// TIA Portal V18 export
VAR_GLOBAL   // PLC tag table "Default tag table"
   CS_Drive_PL_Actor_Interface_AddressIn AT %I50.0 : "PD_TEL105_IN";
   CS_Drive_PL_Actor_Interface_AddressOut AT %Q50.0 : "PD_TEL105_OUT";
   CS_Drive_PP_Actor_Interface_AddressIn AT %I18.0 : "PD_TEL105_IN";
   CS_Drive_PP_Actor_Interface_AddressOut AT %Q18.0 : "PD_TEL105_OUT";
   CS_Drive_TL_Actor_Interface_AddressIn AT %I102.0 : "PD_TEL105_IN";
   CS_Drive_TL_Actor_Interface_AddressOut AT %Q102.0 : "PD_TEL105_OUT";
   CS_Drive_TP_Actor_Interface_AddressIn AT %I76.0 : "PD_TEL105_IN";
   CS_Drive_TP_Actor_Interface_AddressOut AT %Q76.0 : "PD_TEL105_OUT";
   ST23_PAL_Down AT %Q900.0 : Bool;
   ST23_PAL_Up AT %Q900.1 : Bool;
   ST23_MOD1_Up AT %Q900.2 : Bool;
   ST23_MOD2_Up AT %Q900.3 : Bool;
   ST23_MOD3_Up AT %Q900.4 : Bool;
   ST24_PAL_Down AT %Q900.5 : Bool;
   ST24_PAL_Up AT %Q900.6 : Bool;
   ST24_MOD1_Up AT %Q900.7 : Bool;
   ST24_MOD2_Up AT %Q901.0 : Bool;
   ST24_MOD3_Up AT %Q901.1 : Bool;
   ST25_PAL_Down AT %Q901.2 : Bool;
   ST25_PAL_Up AT %Q901.3 : Bool;
   ST25_MOD1_Up AT %Q901.4 : Bool;
   ST25_MOD2_Up AT %Q901.5 : Bool;
   ST25_MOD3_Up AT %Q901.6 : Bool;
   Reserve AT %Q901.7 : Bool;
   ST23_MOD1_Sen11 AT %I900.0 : Bool;
   ST23_MOD1_Sen12 AT %I900.1 : Bool;
   ST23_MOD1_Sen21 AT %I900.2 : Bool;
   ST23_MOD1_Sen22 AT %I900.3 : Bool;
   ST23_MOD2_Sen11 AT %I900.4 : Bool;
   ST23_MOD2_Sen12 AT %I900.5 : Bool;
   ST23_MOD2_Sen21 AT %I900.6 : Bool;
   ST23_MOD2_Sen22 AT %I900.7 : Bool;
   ST23_MOD3_Sen11 AT %I901.0 : Bool;
   ST23_MOD3_Sen12 AT %I901.1 : Bool;
   ST23_MOD3_Sen21 AT %I901.2 : Bool;
   ST23_MOD3_Sen22 AT %I901.3 : Bool;
   ST23_PAL_Sen11 AT %I901.4 : Bool;
   ST23_PAL_Sen12 AT %I901.5 : Bool;
   ST23_PAL_Sen21 AT %I901.6 : Bool;
   ST23_PAL_Sen22 AT %I901.7 : Bool;
   ST24_MOD1_Sen11 AT %I902.0 : Bool;
   ST24_MOD1_Sen12 AT %I902.1 : Bool;
   ST24_MOD1_Sen21 AT %I902.2 : Bool;
   ST24_MOD1_Sen22 AT %I902.3 : Bool;
   ST24_MOD2_Sen11 AT %I902.4 : Bool;
   ST24_MOD2_Sen12 AT %I902.5 : Bool;
   ST24_MOD2_Sen21 AT %I902.6 : Bool;
   ST24_MOD2_Sen22 AT %I902.7 : Bool;
   ST24_MOD3_Sen11 AT %I903.0 : Bool;
   ST24_MOD3_Sen12 AT %I903.1 : Bool;
   ST24_MOD3_Sen21 AT %I903.2 : Bool;
   ST24_MOD3_Sen22 AT %I903.3 : Bool;
   ST24_PAL_Sen11 AT %I903.4 : Bool;
   ST24_PAL_Sen12 AT %I903.5 : Bool;
   ST24_PAL_Sen21 AT %I903.6 : Bool;
   ST24_PAL_Sen22 AT %I903.7 : Bool;
   ST23_Rol_Up AT %Q902.0 : Bool;
   ST24_Rol_Up AT %Q902.1 : Bool;
   ST25_Rol_Up AT %Q902.2 : Bool;
   ST25_MOD1_Sen11 AT %I904.0 : Bool;
   ST25_MOD1_Sen12 AT %I904.1 : Bool;
   ST25_MOD1_Sen21 AT %I904.2 : Bool;
   ST25_MOD1_Sen22 AT %I904.3 : Bool;
   ST25_MOD2_Sen11 AT %I904.4 : Bool;
   ST25_MOD2_Sen12 AT %I904.5 : Bool;
   ST25_MOD2_Sen21 AT %I904.6 : Bool;
   ST25_MOD2_Sen22 AT %I904.7 : Bool;
   ST25_MOD3_Sen11 AT %I905.0 : Bool;
   ST25_MOD3_Sen12 AT %I905.1 : Bool;
   ST25_MOD3_Sen21 AT %I905.2 : Bool;
   ST25_MOD3_Sen22 AT %I905.3 : Bool;
   ST25_PAL_Sen11 AT %I905.4 : Bool;
   ST25_PAL_Sen12 AT %I905.5 : Bool;
   ST25_PAL_Sen21 AT %I905.6 : Bool;
   ST25_PAL_Sen22 AT %I905.7 : Bool;
   "90" AT %Q0.0 : Bool;
   Estop_SS2_ChA AT %I915.0 : Bool;
   Estop_SS2_ChB AT %I915.4 : Bool;
   ST23_25_Y0 AT %Q910.0 : Bool;
   ST23_25_M0 AT %Q910.1 : Bool;
END_VAR
